{attribute addProperty BoxType "AMI8000-0000-0016"}
{attribute addProperty Id "StatuswordAT %I*UINT162"}
{attribute addProperty CRC "1405865676"}
{attribute addProperty SizeInBites "16"}
{attribute addProperty SizeInBytes "2"}
TYPE DRV_Statusword_53CBCECC :
STRUCT
	{attribute addProperty Name "Statusword"}
	Statusword AT %I* : UINT;
END_STRUCT
END_TYPE

(* stored: Version 1.2.0.0, ProductVersion 3.1.4024.9
   DUT DRV_Statusword_53CBCECC: Id {89b5ca27-57e0-4599-879c-5e8ce5e97dcf} *)
